(* CODESYS project cmt251-630.project
   Version: 0.0.0.0
   Title: cmt251-630
   Author: Kleyton

Project tree, tasks and I/O mapping:
  tm251me : TM251MESE, Schneider Electric, order no. TM251MESE, version 5.0.8.2
    application Application
      task MAST (cyclic, interval 20 ms, priority 15, watchdog 100 ms x 1) calls Main_CMD
      global variables GVL
      program Main_CMD [ST]
      RegisterDescription/
        function ETADescription [ST]
        function CMDDescription [ST]
      program Main_Write [ST]
    IO_Bus : IO bus - TM3, Schneider Electric, version 5.0.8.2
    COM_Bus : COM bus, Schneider Electric, version 5.0.8.2
    Ethernet_1 : Ethernet Network, Schneider Electric, version 5.0.8.2
    Ethernet_2 : Device Network, Schneider Electric, version 5.0.8.2
        settings: IPAddress = [192, 168, 100, 50]; SubnetMask = [255, 255, 255, 0]; WebServer = TRUE; FTP Server = FALSE; SoMachine Protocol = TRUE; Modbus Server = TRUE; NetManage Protocol = TRUE; SNMP protocol = FALSE; Enable Routing = FALSE; WebVisu protocol = FALSE; DHCP Server Active = FALSE
      Industrial_Ethernet_Manager : Industrial Ethernet Manager, Schneider Electric, version 1.0.12.31
          settings: BinaryFileSize = 396; Dhcps Host 1.Client Device Name = 'ATV6XX_2'; Dhcps Host 1.Client IP Address = [192, 168, 100, 40]; Dhcps Host 1.Network Mask = [255, 255, 255, 0]; serialized Values = b26d7d7c-3e28-4386-b44d-aa84c393e366=1|; InterfaceUsedByDhcpSize = 4; InterfaceUsedByDhcp = [192,168,100,50]
          unmapped channels: Global Status, Healthbit 0, Healthbit 1, Healthbit 2, Healthbit 3
        Altivar_6xx : Altivar 6••, Schneider Electric, order no. 6••, version 1.1.4.0
            settings: DeviceNumber = 512; Object Input1 = [32, 32, 21233664, 0]; Object Output1 = [33, 32, 25427968, 0]; Default Unit-ID = 248; IPAddress = [192, 168, 100, 40]; ATV6xx channel.Channel ID = 0; ATV6xx channel.Read Offset = 16#0000; ATV6xx channel.Write Offset = 16#0000
            unmapped channels: Statusword, Output speed, InputWord 3, InputWord 4, InputWord 5, InputWord 6, InputWord 7, InputWord 8, InputWord 9, InputWord 10, InputWord 11, InputWord 12, InputWord 13, InputWord 14, InputWord 15, InputWord 16, InputWord 17, InputWord 18, InputWord 19, InputWord 20, InputWord 21, InputWord 22, InputWord 23, InputWord 24, InputWord 25, InputWord 26, InputWord 27, InputWord 28, InputWord 29, InputWord 30, InputWord 31, InputWord 32, Control word, Speed reference, OutputWord 3, OutputWord 4, OutputWord 5, OutputWord 6, OutputWord 7, OutputWord 8,
              OutputWord 9, OutputWord 10, OutputWord 11, OutputWord 12, OutputWord 13, OutputWord 14, OutputWord 15, OutputWord 16, OutputWord 17, OutputWord 18, OutputWord 19, OutputWord 20, OutputWord 21, OutputWord 22, OutputWord 23, OutputWord 24, OutputWord 25, OutputWord 26, OutputWord 27, OutputWord 28, OutputWord 29, OutputWord 30, OutputWord 31, OutputWord 32
    Serial_Line_1 : Serial line, Schneider Electric, version 5.0.8.2
      Machine_Expert_Network_Manager : Machine Expert-Network Manager, Schneider Electric, version 4.0.0.3
  FdtConnections : FDT Connections, Schneider Electric, version 1.0.0.2
*)

// tm251me/Application/GVL
{attribute 'qualified_only'}
VAR_GLOBAL
END_VAR

// tm251me/Application/Main_CMD
PROGRAM Main_CMD
VAR
	
	(*************************************************************)
    (*********** Variáveis para Bloco de Comunicação *************)
    (*************************************************************)
	(* Declaração do Bloco de Comunicação com o inversor *)
	ADDM_atv630Add		:	ADDM;
	(* Variável para identificação do primeiro ciclo *)
	b_firstCycle		:	BOOL	:=	TRUE;
	(* Endereço IP do inversor*)
	s_AddressInv		:	STRING	:=	'192.168.100.40';
	(* Endereço para o cabeçalho do Protocolo *)
	s_AddressInvAll		:	STRING;
	(* Endereço obtido pelo bloco de comunicação *)
	s_AddressModbusTcp	:	ADDRESS;
	
	
	(*************************************************************)
    (********************* Bloco de Pulso ************************)
    (*************************************************************)
	BL_Pulse			:	BLINK;
	
	(*************************************************************)
    (************** Variáveis para Bloco de Pulso ****************)
    (*************************************************************)
	t_High				:	TIME	:=	T#100MS; (* 100 MS para borda alta *)
	t_Low				:	TIME	:=	T#100MS; (* 100MS paea borda baixa *)
	b_Enable			:	BOOL	:=	TRUE;	 (* Habilita bloco de pulso *)
	
	(*************************************************************)
    (************* Variáveis para Bloco de Leitura ***************)
    (*************************************************************)
	(*Bloco de Leitura de dados do equipamento*)
	RV_ETAatv630			:	READ_VAR;
	RV_CMDatv630			:	READ_VAR;
	RV_HMISatv630			:	READ_VAR;
	
	(*************************************************************)
    (************* Variáveis para Bloco de Ecrita ****************)
    (*************************************************************)
	SG_WriteSingleCMDatv630	:	SINGLE_WRITE;
	SG_WriteSingleMotorRot		:	SINGLE_WRITE;
	SG_WriteSingleQuickStop		:	SINGLE_WRITE;
	(*************************************************************)
    (********* Variáveis de análise dos Registradores ************)
    (*************************************************************)
	w_DataReadETAatv630			:	WORD; (* Variável para armazenar dados do registrador ETA *)
	w_DataRCMDatv630			:	WORD; (* Variável para obter os dados do registrador CMD *)
	w_DataWCMDatv630			:	WORD; (* Variável para armazenar dados do registrador CMD *)
	w_QuickStop					:	WORD	:=	2; (* Parada Rápida *)
	i_RotMotoratv630			:	INT; (* Variável para controlar velocidade do motor *)
END_VAR
VAR
	(*************************************************************)
    (****************** Variáveis para debug *********************)
    (*************************************************************)
	b_Pronto					:	BOOL;	(* Variável para colocar dispositivo em Estado de Pronto *)
	b_Energia					:	BOOL;	(* Variável para colocar dispositivo em Estado de Pronto *)
	b_Ligar						:	BOOL;	(* Variável para colocar dispositivo em Estado de Pronto *)
	b_Parar						:	BOOL;	(* Variável para colocar dispositivo em Estado de Pronto *)
	b_Limpar					:	BOOL;	(* Variável para colocar dispositivo em Estado de Pronto *)
	i_Velocidade				:	UINT;	(* Variável para colcoar velocidade do motor *)
END_VAR

(* Verifica se já executou alguma vez *)
IF(b_firstCycle)	THEN
	(* 3 Coloca a comunicação por Ethernet *)
	s_AddressInvAll := CONCAT('3{', s_AddressInv);
	(* 248 é o endereco do equipamento da na rede Ethernet ModBus *)
	s_AddressInvAll	:= CONCAT(s_AddressInvAll,'}248');
END_IF

BL_Pulse(
	ENABLE		:=	b_Enable,
	TIMELOW		:=	t_Low,
	TIMEHIGH	:=	t_High, 
	OUT=>
);

ADDM_atv630Add(
	(*************************  IN/OUT *****************************)
	(* IN_OU Endereço do TCP ModBus *)
	AddrTable	:=	s_AddressModbusTcp,
	(* Varia o Bloco para reconectar novamente *)
	Execute		:=	BL_Pulse.OUT,
	(* Cabeçalho de Endereco para conexão com o equipamento *)
	Addr		:=	s_AddressInvAll,
	(***************************** OUT ******************************)
	(* Informa se a operação ocorreu com sucesso *)
	Done		=>,
	(* Informa se houve erro na comunicação *)
	Error		=>,
	(* Byte para indicar problemas na comunicação *)
	CommError	=>
	);
	
CMDDescription(
	b_Ready		:=	b_Pronto,
	b_Power		:=	b_Energia,
	b_QuickStop	:=	FALSE,
	b_Run		:=	b_Ligar,
	b_Clear		:= 	b_Limpar,
	b_Stop		:=	FALSE,
	w_CMDWord	:=	w_DataWCMDatv630
	);

SG_WriteSingleCMDatv630(
	(* Pronto para executar o Bloco *)
	Execute		:=	ADDM_atv630Add.Done AND NOT ADDM_atv630Add.Error,
	(* Bloco tem de ser executado *)
	Abort		:=	FALSE,
	(* Endereço do bloco ADDM_ModbusTCP_ATVIMC para conexão *)
	Addr		:=	s_AddressModbusTcp,
	(* Tempo Máximo de espera(500ms) *)
	Timeout		:=	5,
	(* Tipo de objeto a ser escrito *)
	ObjType		:=	ObjectType.MW,
	(* Endereco do Objeto a ser escrito *)
	FirstObj	:=	8501,
	(* Palavra a ser escrita *)
	theWord    := w_DataWCMDatv630,
	(* Término da exeução da atividade *)
	Done       => ,
	(* Bloco ainda está ocupado *)
	Busy       => ,
	(* Execução encerrada com exceções *)
	Aborted    => ,
	(* Erro detectados *)
	Error      => ,
	(* Palavra com erros detectados *)
	CommError  => ,
	(* Erros da operação *)
	OperError  =>
	);
	
SG_WriteSingleMotorRot(
	(* Pronto para executar o Bloco *)
	Execute		:=	SG_WriteSingleCMDatv630.Done AND NOT SG_WriteSingleMotorRot.Error AND
			SG_WriteSingleCMDatv630.Done AND NOT SG_WriteSingleCMDatv630.Error,
	(* Bloco tem de ser executado *)
	Abort		:=	FALSE,
	(* Endereço do bloco ADDM_ModbusTCP_ATVIMC para conexão *)
	Addr		:=	s_AddressModbusTcp,
	(* Tempo Máximo de espera(500ms) *)
	Timeout		:=	5,
	(* Tipo de objeto a ser escrito *)
	ObjType		:=	ObjectType.MW,
	(* Endereco do Objeto a ser escrito *)
	FirstObj	:=	8602,
	(* Palavra a ser escrita *)
	theWord    := REAL_TO_WORD(i_RotMotoratv630),
	(* Término da execução da atividade *)
	Done       => ,
	(* Bloco ainda está ocupado *)
	Busy       => ,
	(* Execução encerrada com exceções *)
	Aborted    => ,
	(* Erro detectados *)
	Error      => ,
	(* Palavra com erros detectados *)
	CommError  => ,
	(* Erros da operação *)
	OperError  =>
	);

RV_CMDatv630(
(*************************  IN/OUT *****************************)
(* Verifica se está pronto para leitura *)
Execute		:= ADDM_atv630Add.Done AND NOT ADDM_atv630Add.Error AND
			SG_WriteSingleQuickStop.Done AND NOT SG_WriteSingleQuickStop.Error,
(***************************** IN *******************************)
(* Saída repentina da FB *)
Abort		:=	FALSE,
(* Endereço ModBus para conexão *)
Addr		:=	s_AddressModbusTcp,
(* Tempo Máximo de espera(500ms) *)
Timeout		:=	5,
(* Tipo de Objeto a ser lido *)
ObjType		:=	ObjectType.MW,
(* Início do Objeto a ser lido *)
FirstObj	:=	8501,
(* Quantidade de Endereços lido a partir do primeiro *)
Quantity	:=	1,
(* Aramzenamento do Dado lido remotamente *)
Buffer		:= ADR(w_DataRCMDatv630),
(***************************** OUT ******************************)
(* Conclusão da atividade *)
Done		=>,
(* Bloco ocupado *)
Busy		=>,
(* Execução encerrada com erros *)
Aborted		=>,
(* Erro na operação de leitura da informação *)
Error		=>,
(* Erros detectados na comunicação *)
CommError	=>,
(* Erros detectados na operação *)
OperError	=>	
);

RV_ETAatv630(
(*************************  IN/OUT *****************************)
(* Verifica se está pronto para leitura *)
Execute		:= ADDM_atv630Add.Done AND NOT ADDM_atv630Add.Error,
(***************************** IN *******************************)
(* Saída rependtina da FB *)
Abort		:=	FALSE,
(* Endereço ModBus para conexão *)
Addr		:=	s_AddressModbusTcp,
(* Tempo Máximo de espera(500ms) *)
Timeout		:=	5,
(* Tipo de Objeto a ser lido *)
ObjType		:=	ObjectType.MW,
(* Início do Objeto a ser lido *)
FirstObj	:=	3201,
(* Quantidade de Endereços lido a partir do primeiro *)
Quantity	:=	1,
(* Aramzenamento do Dado lido remotamente *)
Buffer		:= ADR(w_DataReadETAatv630),
(***************************** OUT ******************************)
(* Conclusão da atividade *)
Done		=>,
(* Bloco ocupado *)
Busy		=>,
(* Execução encerrada com erros *)
Aborted		=>,
(* Erro na operação de leitura da informação *)
Error		=>,
(* Erros detectados na comunicação *)
CommError	=>,
(* Erros detectados na operação *)
OperError	=>	
);



IF((NOT RV_ETAatv630.Busy AND RV_ETAatv630.Done AND NOT RV_ETAatv630.Error) OR TRUE) THEN
ETADescription(
(***************************** IN *******************************)
(* Entrada da palavra obtida do Registrador *)
w_ETARegister	:=	w_DataReadETAatv630,
(***************************** OUT ******************************)
b_PowerReady	=>,
b_Ready			=>,
b_Enable		=>,
b_Fail			=>,
b_Voltage_On	=>,
b_QuickStop		=>,
b_PowerBlocked	=>,
b_Warning		=>,
b_CmtFieldBus	=>,
b_RefSpeed		=>,
b_LimitActive	=>,
b_StopKey		=>,
b_Direction		=>);
END_IF

	
b_firstCycle := FALSE;

END_PROGRAM

// tm251me/Application/RegisterDescription/CMDDescription
(************************************************************)
(***** Registrador CMD no ATV6xx são registradores para *****)
(** Prepara o Inversor o inversor para partir e colocar o ***)
(******************* Motor para rodar ***********************)
(************************************************************)
FUNCTION CMDDescription : BOOL
VAR_INPUT
    b_Ready     :   BOOL; (* Coloca o inversor em prontidão para Acionamento do Motor *)
    b_Power     :   BOOL; (* Seleciona Alimentação para o motor *)
	b_QuickStop	:	BOOL; (* Parada Rápida *)
	b_Run		:	BOOL; (* Acionamneto do Motor *)
	b_Clear		:	BOOL; (* Comando de Rearm do Motor *)
	b_Stop		:	BOOL; (* Comando de para do Motor( Será utilizada parada configurada no registrador STT ). *)
END_VAR
VAR_IN_OUT
	w_CMDWord	:	WORD; (* Palavra do conteúdo do Registrador lido / Mudança das posições conforme configuração dos bits *)
END_VAR
VAR
END_VAR

w_CMDWord.0		:=	b_Run;
w_CMDWord.1		:=	b_Power;
w_CMDWord.2		:=	b_QuickStop;
w_CMDWord.3 	:=	b_Ready;
w_CMDWord.7		:=	b_Clear;
w_CMDWord.8		:=	b_Stop;

END_FUNCTION

// tm251me/Application/RegisterDescription/ETADescription
FUNCTION ETADescription : BOOL
VAR_INPUT
	w_ETARegister	:	WORD;	(* Palavra de entrada para a função *)
END_VAR
VAR
END_VAR
VAR_OUTPUT
	b_PowerReady	:	BOOL;	(* Dispositivo alimentado *)
	b_Ready			:	BOOL;	(* Dispositivo pronto para Ligar Motor *)
	b_Enable		:	BOOL;	(* Dispositivo em Execução *)
	b_Fail			:	BOOL;	(* Detectado falha no dispositivo *)
	b_Voltage_On	:	BOOL;	(* Alimentação conectada (TRUE) / Não comentada (FALSE) *)
	b_QuickStop		:	BOOL;	(* Motor parado usando método rápido *)
	b_PowerBlocked	:	BOOL;	(* Alimentação Bloqueada *)
	b_Warning		:	BOOL;	(* Detectado Alertas *)
	b_CmtFieldBus	:	BOOL;	(* Referência via fieldbus *)
	b_RefSpeed		:	BOOL;	(* Referência de velocidade quando motor está rodando *)
	b_LimitActive	:	BOOL;	(* 0 - A referência  do motor esta dentro dos limites LSB e HSP / 1 - Limite estrapolado *)
	b_StopKey		:	BOOL;	(* Botão de parada na IHM *)
	b_Direction		:	BOOL;	(* 0 - Rotação com direção para frente / 1 - Rotação com direção para trás *)
END_VAR

(*************************************************************)
(*** Identificação dos bits para Erros a partir do Reg ETA ***)
(*************************************************************)
b_PowerReady	:=	w_ETARegister.0;
b_Ready			:=	w_ETARegister.1;
b_Enable		:=	w_ETARegister.2;
b_Fail			:=	w_ETARegister.3;
b_Voltage_On	:=	w_ETARegister.4;
b_QuickStop		:=	w_ETARegister.5;
b_PowerBlocked	:=	w_ETARegister.6;
b_Warning		:=	w_ETARegister.7;
b_CmtFieldBus	:=	w_ETARegister.9;
b_RefSpeed		:=	w_ETARegister.10;
b_LimitActive	:=	w_ETARegister.11;
b_StopKey		:=	w_ETARegister.14;
b_Direction		:=	w_ETARegister.15;

END_FUNCTION

// tm251me/Application/Main_Write
PROGRAM Main_Write
VAR
	
	(*************************************************************)
    (*********** Variáveis para Bloco de Comunicação *************)
    (*************************************************************)
	(* Declaração do Bloco de Comunicação com o inversor *)
	ADDM_atv630Add		:	ADDM;
	(* Variável para identificação do primeiro ciclo *)
	b_firstCycle		:	BOOL	:=	TRUE;
	(* Endereço IP do inversor*)
	s_AddressInv		:	STRING	:=	'192.168.100.40';
	(* Endereço para o cabeçalho do Protocolo *)
	s_AddressInvAll		:	STRING;
	(* Endereço obtido pelo bloco de comunicação *)
	s_AddressModbusTcp	:	ADDRESS;
	
	(*************************************************************)
    (************* Variáveis para Bloco de Leitura ***************)
    (*************************************************************)
	(*Bloco de Leitura de dados do equipamento*)
	RV_ETAatv630			:	READ_VAR;
	RV_CMDatv630			:	READ_VAR;
	
	(*************************************************************)
    (************* Variáveis para Bloco de Ecrita ****************)
    (*************************************************************)
	SG_WriteSingleCMDagtv630	:	SINGLE_WRITE;
	(*************************************************************)
    (********* Variáveis de análise dos Registradores ************)
    (*************************************************************)
	w_DataReadETAatv630		:	WORD; (* Variável para armazenar dados do registrador ETA *)
	w_DataRCMDatv630		:	WORD; (* Variável para obter os dados do registrador CMD *)
	w_DataWCMDatv630		:	WORD; (* Variável para armazenar dados do registrador CMD *)
END_VAR

IF(b_firstCycle)	THEN
	(* 3 Coloca a comunicação por Ethernet *)
	s_AddressInvAll := CONCAT('3{', s_AddressInv);
	(* 248 é o endereco do equipamento da na rede Ethernet ModBus *)
	s_AddressInvAll	:= CONCAT(s_AddressInvAll,'}248');
END_IF

ADDM_atv630Add(
	(*************************  IN/OUT *****************************)
	(* IN_OUT Endereço do TCP ModBus *)
	AddrTable	:=	s_AddressModbusTcp,
	(* Trata o Bloco e informa que a configuração já foi executada uma vez*)
	Execute		:=	NOT b_firstCycle,
	(* Cabeçalho de Endereco para conexão com o equipamento *)
	Addr		:=	s_AddressInvAll,
	(***************************** OUT ******************************)
	(* Informa se a operação ocorreu com sucesso *)
	Done		=>,
	(* Informa se houve erro na comunicação *)
	Error		=>,
	(* Byte para indicar problemas na comunicação *)
	CommError	=>
	);

w_DataWCMDatv630	:=	0;
		CMDDescription(
			b_Ready		:=	TRUE,
			b_Power		:=	TRUE,
			b_QuickStop	:=	FALSE,
			b_Run		:=	TRUE,
			b_Clear		:= 	FALSE,
			b_Stop		:=	FALSE,
			w_CMDWord	:=	w_DataWCMDatv630
			);

SG_WriteSingleCMDagtv630(
			(* Pronto para executar o Bloco *)
			Execute		:=	ADDM_atv630Add.Done AND NOT ADDM_atv630Add.Error,
			(* Bloco tem de ser executado *)
			Abort		:=	FALSE,
			(* Endereço do bloco ADDM_ModbusTCP_ATVIMC para conexão *)
			Addr		:=	s_AddressModbusTcp,
			(* Tempo Máximo de espera(500ms) *)
			Timeout		:=	5,
			(* Tipo de objeto a ser escrito *)
			ObjType		:=	ObjectType.MW,
			(* Endereco do Objeto a ser escrito *)
			FirstObj	:=	8501,
			(* Palavra a ser escrita *)
			theWord    := w_DataWCMDatv630,
			(* Término da exeução da atividade *)
			Done       => ,
			(* Bloco ainda está ocupado *)
			Busy       => ,
			(* Execução encerrada com exceções *)
			Aborted    => ,
			(* Erro detectados *)
			Error      => ,
			(* Palavra com erros detectados *)
			CommError  => ,
			(* Erros da operação *)
			OperError  =>
			);
			
b_firstCycle	:=		FALSE;

END_PROGRAM
